PROGRAM Stn052_41_Stn124MainMergePrestop
VAR
	//correct
	{attribute 'TcLinkToOSO' := '.iPuckPresent    :=  <0,1,2>TIIB[N27S00 (AL1332)]^N27S03 (AL2341)^TxPDO^input byte 1;
								 .iBufferFull   :=  <0,1,2>TIIB[N27S00 (AL1332)]^N27S03 (AL2341)^TxPDO^input byte 3;
								 .oStopLower    :=  <0,1,1>TIIB[N27S00 (AL1332)]^N27S06 (EX260)^RxPDO^output byte 1'}	
	fbConvStop: FB_ConvStop;
END_VAR

//  This code instantiates a component that is implimented as a common function block
//    Note that I/O is linked directly to I/O variables inside the named instance

gStn052_41_Stn124MainMergePrestop.ConvRunning := gConsumed_SafetyInterfaceConv.MtrRunning.Enc054Mtr05;

fbConvStop(
	pStn := ADR(gStn052),
	pCmp := ADR(gStn052_41_Stn124MainMergePrestop),
	pUpstreamStop := 0,
	pStateTraceBuffer := ADR(gStn052_StateTraceBuffer),
	pStateTraceFifo := ADR(gStn052_StateTraceFifo),
	pStats := ADR(gStn052_02_Stats));

END_PROGRAM

(* stored: Version 1.1.0.1, ProductVersion 3.1.4024.6
   POU Stn052_41_Stn124MainMergePrestop: Id {9010e723-0279-48da-a19f-fbc3ee4756b4}, SpecialFunc None *)
